TYPE csp_main_accuChange_partColor_enum :
(
	NO_COLOR		 	:= 0,
	RED					:= 1,
	GREEN				:= 2,
	BLUE				:= 3,
	YELLOW				:= 4,
	WHITE				:= 5,
	BLACK				:= 6,
	ORANGE				:= 7
);
END_TYPE

(* stored: Version 1.1.0.1, ProductVersion 3.1.4022.18
   DUT csp_main_accuChange_partColor_enum: Id {eb654986-f064-4a0f-9bca-c4c85ecd528c} *)
